Staubli VAL3: init.pgx

program init(num x_nEncNum, string x_sTask)
begin
  //
  //***************************
  //***** Numerical value *****
  //***************************
  nPresetPos=0
  // -- Max value of encoder device input in counts:
  // considering a internal counter unsigned 32 bits
  nMAXCOUNT=power(2,32)
  nMINCOUNT=0
  //
  //***************************
  //********* Strings *********
  //***************************
  sTASK=x_sTask+toString("",x_nEncNum)
  sEncNum="ENC"+toString("",x_nEncNum)
  //
  //***************************
  //* INITIALIZATION  SECTION *
  //***************************
  //-- Detection of rising edge on encoder latch input
  bMemoLatchState=diEncLatched
  //-- Select if position capture INPUT occurs on rising/falling edge
  //   bLatchLevel=true --> position capture on rising edge
  //   bLatchLevel=false --> position capture on falling edge
  //        if position capture OUTPUT occurs on falling edge
  //        CHANGE the logic of the output (doClock=false --> true)
  //        in the program conveyor of the conveyor lib
  bLatchLevel=true
  //-- Part has been latched
  bPartLatched=false
  //
  // Preset encoder counter
  aioSet(aoPresetPos,nPresetPos)
  doEnablePreset=true
  //
  // Reset latch register
  doEnableLatch=false
  // Initialize encoder values
  nEncLatchedVal=nEncValue=0
  //
  bLatchEnabled=true
end
